// TwinCAT 3 PLC project _04_ChainOfResponsibility
// ProgramVersion: 3.1.4023.0
// libraries:
//   Tc2_Standard, * (Beckhoff Automation GmbH)
//   Tc2_System, * (Beckhoff Automation GmbH)
//   Tc3_Module, * (Beckhoff Automation GmbH)
// project tree:
//   Chain Of Responsibility Pattern/Handlers/ FB_BaseHandler.TcPOU, FB_StaticHandler1.TcPOU, FB_StaticHandler2.TcPOU, FB_StaticHandler3.TcPOU, FB_StaticHandler_n.TcPOU, I_Handler.TcIO
//   Chain Of Responsibility Pattern/ P_ChainOfResponsibility.TcPOU
//   / MAIN.TcPOU, PlcTask.TcTTO
// (motion and I/O tree: see PLC project 13_decorator)
// real-time tasks:
//   TASK PlcTask: cycle T#10ms, priority 20, ADS port 350
// variable links:

CONFIGURATION _04_ChainOfResponsibility
    RESOURCE PLC ON TwinCAT3
        TASK PlcTask(INTERVAL := T#10ms, PRIORITY := 20);
        PROGRAM MAIN WITH PlcTask : MAIN;
    END_RESOURCE
END_CONFIGURATION

// ---- Chain Of Responsibility Pattern/Handlers/I_Handler.TcIO
INTERFACE I_Handler

METHOD handle : BOOL
VAR_INPUT
	request	:	STRING;
END_VAR
END_METHOD

METHOD setNext : BOOL
VAR_INPUT
	h	: I_Handler;
END_VAR
END_METHOD

END_INTERFACE

// ---- MAIN.TcPOU
PROGRAM MAIN
VAR
END_VAR

(* 
	GOF 		Avoid coupling the sender of a request to its receiver by giving more than one
				object the chance to handle the request. Chain the receiving objects and pass 
				the request along the chain until an object handles it    
*)
P_ChainOfResponsibility();

END_PROGRAM

// ---- Chain Of Responsibility Pattern/P_ChainOfResponsibility.TcPOU
// Copyright (c) 2021, John Helfrich
PROGRAM P_ChainOfResponsibility
VAR
	h1				:	FB_StaticHandler1;
	h2				:	FB_StaticHandler2;
	h3				:	FB_StaticHandler3;
	h_n				:	FB_StaticHandler_n;
	request 		:	STRING	:= 'Hello world!';
	xStartProcess	: 	BOOL;
END_VAR

h1.setNext(h2);
h2.setNext(h3);
h3.setNext(h_n);

(*************************************************************
*************SIMULATION***************************************
***
*** Leave request as "hello world!" for full chain processing
*** or use the string phrases below to interupt the chain.
***
***	Handler 1 - request := 'Handler 1 Interupt';
*** Handler 2 - request := 'Handler 2 Interupt';
*** Handler 3 - request := 'Handler 3 Interupt';
**************************************************************
*************************************************************)

IF xStartProcess THEN
	xStartProcess := FALSE;
	h1.handle(request);
END_IF

END_PROGRAM

// ---- Chain Of Responsibility Pattern/Handlers/FB_StaticHandler1.TcPOU
FUNCTION_BLOCK FB_StaticHandler1 EXTENDS FB_BaseHandler
VAR_INPUT
END_VAR
VAR_OUTPUT
END_VAR
VAR
END_VAR

METHOD handle : BOOL
VAR_INPUT
	request	:	STRING;
END_VAR
IF request = 'Handler 1 Interupt' THEN
	ADSLOGSTR(ADSLOG_MSGTYPE_MSGBOX, request, ' ');
ELSE
	ADSLOGSTR(ADSLOG_MSGTYPE_MSGBOX, '@H1 Moving to next handler ', '');
	SUPER^.handle(request);
END_IF
END_METHOD

END_FUNCTION_BLOCK

// ---- Chain Of Responsibility Pattern/Handlers/FB_BaseHandler.TcPOU
FUNCTION_BLOCK FB_BaseHandler IMPLEMENTS I_Handler
VAR_INPUT
END_VAR
VAR_OUTPUT
END_VAR
VAR
	next : I_Handler;
END_VAR

METHOD handle : BOOL
VAR_INPUT
	request	:	STRING;
END_VAR
IF ADR(next) <> 0 THEN
	next.handle(request);
END_IF
END_METHOD

METHOD setNext : BOOL
VAR_INPUT
	h	: I_Handler;
END_VAR
next := h;
END_METHOD

END_FUNCTION_BLOCK

// ---- Chain Of Responsibility Pattern/Handlers/FB_StaticHandler2.TcPOU
FUNCTION_BLOCK FB_StaticHandler2 EXTENDS FB_BaseHandler
VAR_INPUT
END_VAR
VAR_OUTPUT
END_VAR
VAR
END_VAR

METHOD handle : BOOL
VAR_INPUT
	request	:	STRING;
END_VAR
IF request = 'Handler 2 Interupt' THEN
	ADSLOGSTR(ADSLOG_MSGTYPE_MSGBOX, request, ' ');
ELSE
	ADSLOGSTR(ADSLOG_MSGTYPE_MSGBOX, '@H2 Moving to next handler ', '');
	SUPER^.handle(request);
END_IF
END_METHOD

END_FUNCTION_BLOCK

// ---- Chain Of Responsibility Pattern/Handlers/FB_StaticHandler3.TcPOU
FUNCTION_BLOCK FB_StaticHandler3 EXTENDS FB_BaseHandler
VAR_INPUT
END_VAR
VAR_OUTPUT
END_VAR
VAR
END_VAR

METHOD handle : BOOL
VAR_INPUT
	request	:	STRING;
END_VAR
IF request = 'Handler 3 Interupt' THEN
	ADSLOGSTR(ADSLOG_MSGTYPE_MSGBOX, request, ' ');
ELSE
	ADSLOGSTR(ADSLOG_MSGTYPE_MSGBOX, '@H3 Moving to next handler ', '');
	SUPER^.handle(request);
END_IF
END_METHOD

END_FUNCTION_BLOCK

// ---- Chain Of Responsibility Pattern/Handlers/FB_StaticHandler_n.TcPOU
FUNCTION_BLOCK FB_StaticHandler_n EXTENDS FB_BaseHandler
VAR_INPUT
END_VAR
VAR_OUTPUT
END_VAR
VAR
END_VAR

METHOD handle : BOOL
VAR_INPUT
	request	:	STRING;
END_VAR
ADSLOGSTR(ADSLOG_MSGTYPE_MSGBOX, request , '');
END_METHOD

END_FUNCTION_BLOCK
